FUNCTION_BLOCK PUBLIC FB_NewEngine EXTENDS FB_Engine
VAR_INPUT
	nGear		:	INT := 2;
	fVelocity	:	LREAL := 8.0;
END_VAR
VAR
	gearInternal		:	INT;
END_VAR

{attribute 'monitoring' := 'variable'}
PROPERTY PUBLIC Gear : INT
GET
Gear := gearInternal;
END_GET
SET
gearInternal := Gear;
END_SET
END_PROPERTY

METHOD PUBLIC Start
VAR_INPUT
	nGear		:	INT := 2;
	fVelocity	:	LREAL := 8.0;
END_VAR
SUPER^.Start(nGear, fVelocity);
Gear := nGear;
END_METHOD

END_FUNCTION_BLOCK

(* stored: Version 1.1.0.1, ProductVersion 3.1.4020.12
   POU FB_NewEngine: Id {02831598-4827-4a85-86c1-fc3eee11db63}, SpecialFunc None
   Property Gear: Id {b1007588-fa86-4c5d-a5f7-94ec3322c92d}
   Get Get: Id {ebd6f5ce-c79c-44c6-80f7-8307ec620339}
   Set Set: Id {1d27ec8f-7fbe-4e19-ada8-caaba952686c}
   Method Start: Id {e96a3668-413d-4934-80e9-328bd8763976} *)
